FUNCTION_BLOCK CentralController (* Basic Function Block Type *)
  (* Standard: 61499-2 *)
  (* Version 0.0, 17/09/2012, spat251, nxtControl GmbH, Template *)
  PACKAGE Main;
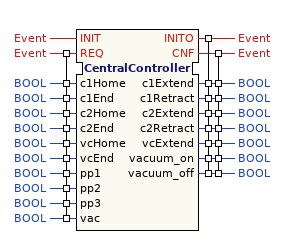
  EVENT_INPUT
    INIT; (* Initialization Request *)
    REQ WITH c1Home, c1End, c2Home, c2End, vcHome, vcEnd, pp1, pp2, pp3, vac; (* Normal Execution Request *)
  END_EVENT
  EVENT_OUTPUT
    INITO WITH c1Extend, vacuum_on, vcExtend, c2Retract, c2Extend, c1Retract, vacuum_off; (* Initialization Confirm *)
    CNF WITH vacuum_on, vcExtend, c2Retract, c2Extend, c1Retract, c1Extend, vacuum_off; (* Execution Confirmation *)
  END_EVENT
  VAR_INPUT
    c1Home : BOOL; (* Input event qualifier *)
    c1End : BOOL;
    c2Home : BOOL;
    c2End : BOOL;
    vcHome : BOOL;
    vcEnd : BOOL;
    pp1 : BOOL;
    pp2 : BOOL;
    pp3 : BOOL;
    vac : BOOL;
  END_VAR
  VAR_OUTPUT
    c1Extend : BOOL; (* Output event qualifier *)
    c1Retract : BOOL;
    c2Extend : BOOL;
    c2Retract : BOOL;
    vcExtend : BOOL;
    vacuum_on : BOOL;
    vacuum_off : BOOL;
  END_VAR
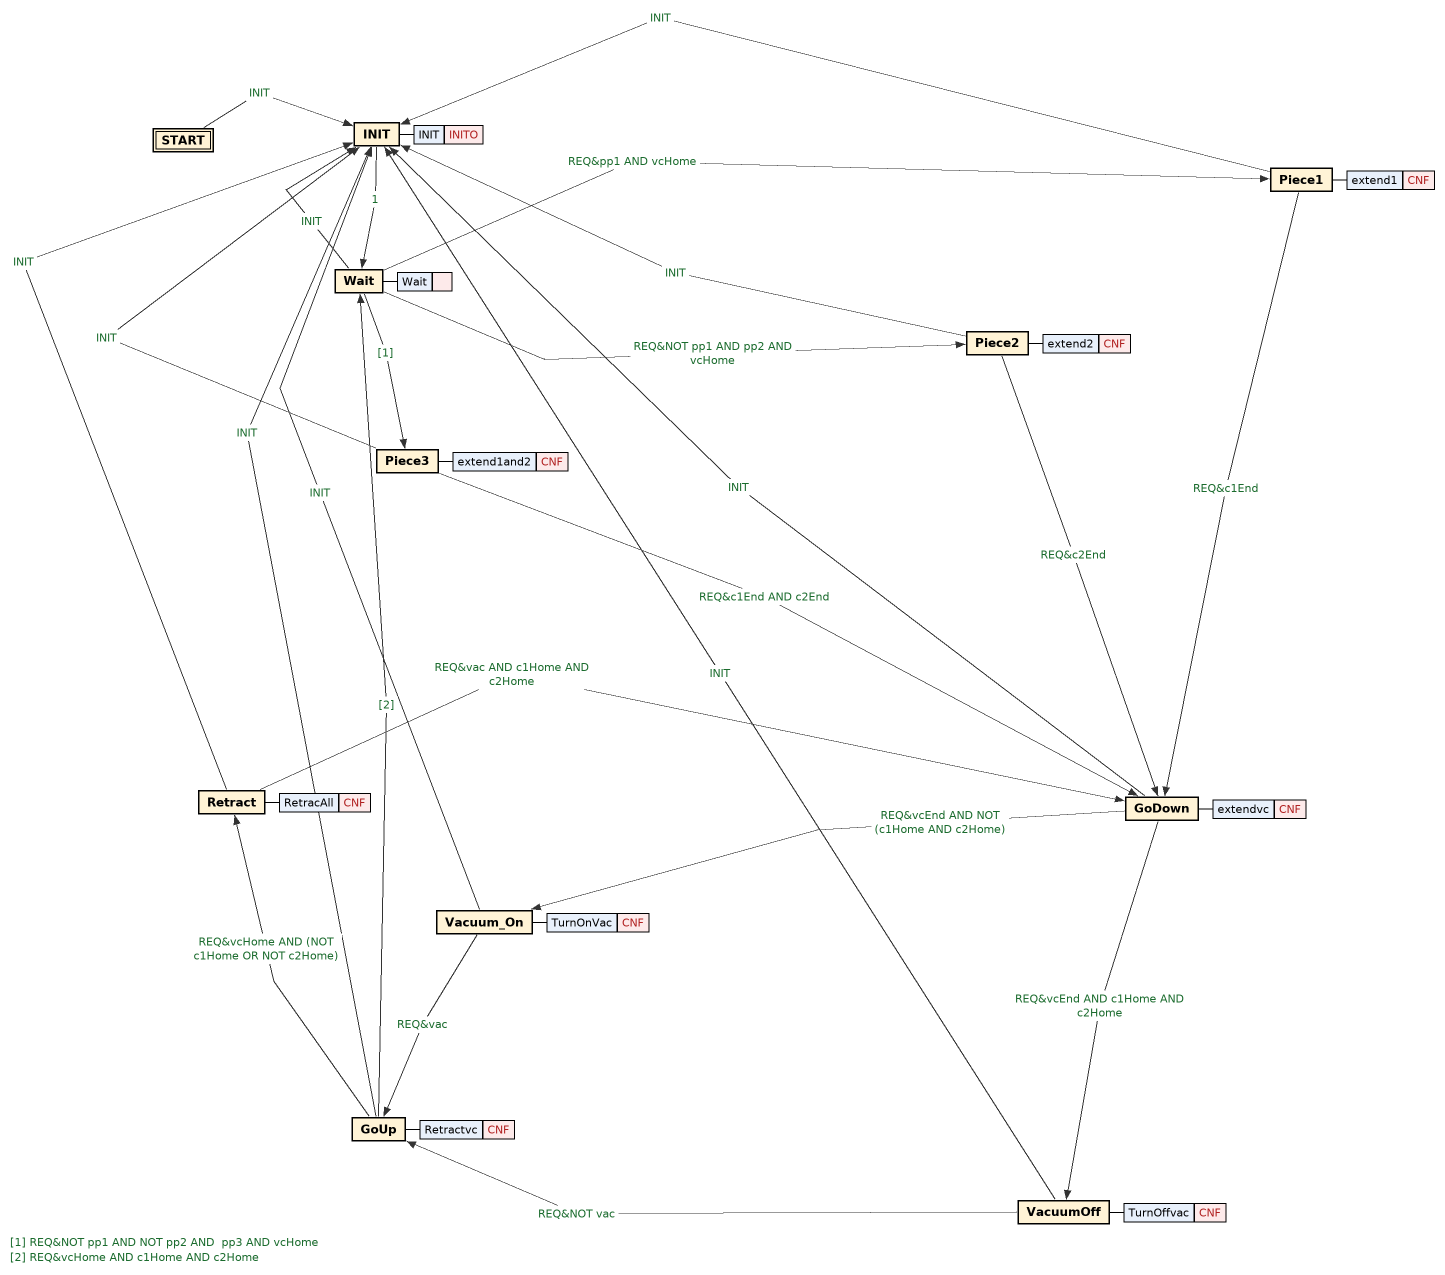
  EC_STATES
    START; (* Initial State *)
    INIT : INIT -> INITO; (* Initialization *)
    GoDown : extendvc -> CNF; (* Normal execution *)
    Wait : Wait;
    Piece1 : extend1 -> CNF;
    Piece2 : extend2 -> CNF;
    Piece3 : extend1and2 -> CNF;
    Vacuum_On : TurnOnVac -> CNF;
    GoUp : Retractvc -> CNF;
    VacuumOff : TurnOffvac -> CNF;
    Retract : RetracAll -> CNF;
  END_STATES
  EC_TRANSITIONS
    START TO INIT := INIT;
    INIT TO Wait := 1;
    GoUp TO Wait := REQ&vcHome AND c1Home AND c2Home;
    Retract TO GoDown := REQ&vac AND c1Home AND c2Home;
    Wait TO Piece1 := REQ&pp1 AND vcHome;
    Wait TO Piece2 := REQ&NOT pp1 AND pp2 AND vcHome;
    Wait TO Piece3 := REQ&NOT pp1 AND NOT pp2 AND  pp3 AND vcHome;
    Piece1 TO GoDown := REQ&c1End;
    Piece2 TO GoDown := REQ&c2End;
    Piece3 TO GoDown := REQ&c1End AND c2End;
    GoDown TO Vacuum_On := REQ&vcEnd AND NOT (c1Home AND c2Home);
    Vacuum_On TO GoUp := REQ&vac;
    VacuumOff TO GoUp := REQ&NOT vac;
    GoDown TO VacuumOff := REQ&vcEnd AND c1Home AND c2Home;
    GoUp TO Retract := REQ&vcHome AND (NOT c1Home OR NOT c2Home);
    Wait TO INIT := INIT;
    Piece1 TO INIT := INIT;
    Piece2 TO INIT := INIT;
    Piece3 TO INIT := INIT;
    Retract TO INIT := INIT;
    Vacuum_On TO INIT := INIT;
    GoDown TO INIT := INIT;
    GoUp TO INIT := INIT;
    VacuumOff TO INIT := INIT;
  END_TRANSITIONS
  ALGORITHM INIT IN ST: (* Initialization algorithm *)
INIT:=FALSE;
c1Extend:=FALSE;
c2Extend:=FALSE;
vcExtend:=FALSE;
c1Retract:=FALSE;
c2Retract:=FALSE;
vacuum_on:=FALSE;
vacuum_off:=FALSE;
  END_ALGORITHM
  ALGORITHM REQ IN ST: (* Normally executed algorithm *)
;
  END_ALGORITHM
  ALGORITHM extend1 IN ST:
c1Extend:=TRUE;
REQ:=FALSE;
  END_ALGORITHM
  ALGORITHM extend2 IN ST:
c2Extend:=TRUE;
REQ:=FALSE;
  END_ALGORITHM
  ALGORITHM extend1and2 IN ST:
c1Extend:=TRUE;
c2Extend:=TRUE;
REQ:=FALSE;
  END_ALGORITHM
  ALGORITHM extendvc IN ST:
vcExtend:=TRUE;
REQ:=FALSE;
  END_ALGORITHM
  ALGORITHM TurnOnVac IN ST:
vacuum_on:=TRUE;
vacuum_off:=FALSE;
REQ:=FALSE;
  END_ALGORITHM
  ALGORITHM Retractvc IN ST:
vcExtend:=FALSE;
REQ:=FALSE;
  END_ALGORITHM
  ALGORITHM TurnOffvac IN ST:
vacuum_on:=FALSE;
vacuum_off:=TRUE;
REQ:=FALSE;
  END_ALGORITHM
  ALGORITHM RetracAll IN ST:
c1Extend:=FALSE;
c2Extend:=FALSE;
c1Retract:=TRUE;
c2Retract:=TRUE;
REQ:=FALSE;
  END_ALGORITHM
  ALGORITHM Wait IN ST:
c1Extend:=FALSE;
c2Extend:=FALSE;
vcExtend:=FALSE;
c1Retract:=FALSE;
c2Retract:=FALSE;
vacuum_on:=FALSE;
vacuum_off:=FALSE;
REQ:=FALSE;
  END_ALGORITHM
END_FUNCTION_BLOCK
